INTERFACE IEvent

METHOD AddEventHandler : IEvent
VAR_INPUT
    Handler : IEventHandlerBase;
END_VAR
END_METHOD

METHOD ClearEventHandlers : IEvent
VAR_INPUT
END_VAR
END_METHOD

END_INTERFACE

(* stored: Version 1.1.0.1, ProductVersion 3.1.4024.3
   Itf IEvent: Id {76b46dd0-9b8c-40e6-9cc2-a8255b4b6f41}
   Method AddEventHandler: Id {f96d4406-f2e0-4ebc-922f-38b4276ed8b0}
   Method ClearEventHandlers: Id {4aa8fa4f-350a-4761-929a-75af37e8488f} *)
